FUNCTION_BLOCK InterpolateNewton
VAR_INPUT
	EN: BOOL;
	x: LREAL;
END_VAR
VAR_OUTPUT
	ENO: BOOL;
	y: LREAL;
END_VAR
VAR CONSTANT
	NUM_POINTS: INT := 9;
END_VAR
VAR
	InitDone: BOOL;
	yd: ARRAY [0..NUM_POINTS - 1, 0..NUM_POINTS - 1] OF LREAL;
	i: INT;
END_VAR
VAR PERSISTENT
	xd: ARRAY [0..NUM_POINTS - 1] OF LREAL;
	yv: ARRAY [0..NUM_POINTS - 1] OF LREAL;
END_VAR

IF NOT InitDone THEN
	FOR i := 0 TO NUM_POINTS - 1 DO
		yd[i, 0] := yv[i];
	END_FOR
	DividedDiffTable();
	InitDone := TRUE;
END_IF
y := ApplyFormula(x);
ENO := EN;

METHOD ApplyFormula : LREAL
VAR_INPUT
	Value: LREAL;
END_VAR
VAR
	Sum: LREAL;
	i: INT;
END_VAR
Sum := yd[0, 0];
FOR i := 1 TO NUM_POINTS - 1 DO
	Sum := Sum + ProTerm(i, Value) * yd[0, i];
END_FOR
ApplyFormula := Sum;
END_METHOD

METHOD DividedDiffTable : BOOL
VAR_INPUT
END_VAR
VAR
	i: INT;
	j: int;
END_VAR
FOR i := 1 TO NUM_POINTS - 1 DO
	FOR j := 0 TO NUM_POINTS - i - 1 DO
		IF ABS(xd[j] - xd[i + j]) > 0.00000001 THEN
			yd[j,i] := (yd[j,i - 1] - yd[j + 1,i - 1]) / (xd[j] - xd[i + j]);			
		END_IF
	END_FOR
END_FOR
DividedDiffTable := TRUE;
END_METHOD

METHOD ProTerm : LREAL
VAR_INPUT
	i: INT;
	Value: LREAL;
END_VAR
VAR
	Pro: LREAL;
	j: int;
END_VAR
Pro := 1;
FOR j := 0 TO i - 1 DO
	Pro := Pro * (Value - xd[j]);
END_FOR
ProTerm := Pro;
END_METHOD

END_FUNCTION_BLOCK

(* stored: Version 1.1.0.1, ProductVersion 3.1.4024.3
   POU InterpolateNewton: Id {b5818b84-20d3-40eb-9693-6144dbb836a6}, SpecialFunc None
   Method ApplyFormula: Id {37dced75-6cd7-4655-9076-4916c1ae9ceb}
   Method DividedDiffTable: Id {efdf09d8-3613-4a4a-8a0f-b90ef3dfcba2}
   Method ProTerm: Id {d2c1070f-e0f4-4c9a-b7f5-b8b4cfe03957} *)
